(* IEC 61131-3 sources: moqui-plc/agent-skills/output/sessions/demo-plant-session/generated-plc/demo-hvac/src/main/org/moqui/device, 4 files *)

(* ---- DeviceFacade.dut ---- *)
(*
 * DeviceFacade implementation for managing devices and logical parameters.
 *
 * Naming rules:
 *   deviceName + parameterName or parameterName -> logical signal
 *   deviceName + parameterName or parameterName + Min/Max -> limits
 *
 * All digital signals (boolean) are active-high (positive logic).
 * All durations are expressed in seconds TUnit.
 *)
TYPE DeviceFacade : STRUCT
    (* ========== Analog process/environment parameters ========== *)
    (* TODO: declare REAL process/environment parameters *)

    (* ========== Digital process/environment parameters ========== *)
    (* TODO: declare BOOL process/environment parameters *)

    (* Boolean predicates - computed each scan by MainRuleEngine *)
    (* TODO: declare computed predicates used by MainRuleEngine *)

    (* Operating-mode flags and process timing (mapped from recipe). *)
    estimatedRuntime : TUnit;
    minRuntime : TUnit;
    estimatedBreakDuration : TUnit;
    minBreakDuration : TUnit;
    processEstimatedDuration : TUnit;
    processMinDuration : TUnit;
    processActualDuration : TUnit;
    processRemainingDuration : TUnit;
    actualRuntime : TUnit;
    actualBreakDuration : TUnit;
    timeBreakEnabled : BOOL;
    isCompleted : BOOL;

    (* Main FSM state and transition request/acknowledge commands *)
    status : MainStatus := MainStatus.Disabled;
    lastStatus : MainStatus := MainStatus.Disabled;
    disabledRequest : BOOL;
    standstillRequest : BOOL;
    homingRequest : BOOL;
    runRequest : BOOL;
    synchronizedRunRequest : BOOL;
    stoppingRequest : BOOL;
    errorStopRequest : BOOL;
    faultRequest : BOOL;
    faultAck : BOOL;

    (* ========== Atomic devices ========== *)
    (* TODO: declare Actuator/ActuatorGroup/Axis/AxisGroup/ProcessPid instances *)

    (* Signal management - centralised fault / alarm / warning engine *)
    signalMgmt : SignalMgmt;
END_STRUCT END_TYPE

(* Questions for the skill/user:
 * 1. Which analog input signals and setpoints must be declared as REAL?
 * 2. Which digital signals must be declared as BOOL?
 * 3. Which computed predicates are required by MainRuleEngine?
 * 4. Which timing/process flags are needed (estimatedRuntime, minRuntime, etc.)?
 * 5. Which request flags correspond to the states in the selected StatusFlow?
 * 6. Which atomic devices exist: Actuator, ActuatorGroup, Axis, AxisGroup, ProcessPid?
 *)

(* ---- IOFacade.dut ---- *)
(*
 * IOFacade implementation for managing physical devices and input/output signals/terminals.
 * Input/Output physical terminals naming rules.
 * From each value of the Parameter entity 3 signals will be generated, according to the following naming convention:
 *     deviceName + parameterName or parameterName + physicalAddress (e.g.: Channel + PhysicalAddress for Modbus)
 *     deviceName + parameterName or parameterName + Min/Max + physicalAddress (e.g.: Channel + PhysicalAddress for Modbus)
 *
 * The physicalAdddress suffix will have the following syntax:
 *    %<memory area prefix> ( <size prefix> )? <memory position>
 * where
 *    <memory area prefix> : I | Q | M
 *    <size prefix> : X | B | W | D
 *    <memory position> : <number> ( .<number> )* (* Depends on the target system *)
 *
 * An alternative is to use semantic signal naming rules.
 *)
TYPE IOFacade : STRUCT
    (* ========== Phyisical Input Terminals/Signals ========== *)
    (* TODO: declare physical input signals from DeviceRequestItem or naming convention *)

    (* ========== Phyisical Output Terminals/Signals ========== *)
    (* TODO: declare physical output signals from DeviceRequestItem or naming convention *)
END_STRUCT END_TYPE

(* Generation notes:
 * - This file is auto-generable from DeviceRequestItem metadata or from naming conventions.
 * - The logical-to-physical mapping remains outside this template and stays manual in V1.
 *
 * Questions for the skill/user:
 * 1. Should names come from DeviceRequestItem.requestItemName or from naming conventions?
 * 2. Which physical signals are inputs and which are outputs?
 * 3. What IEC type should be used for each signal?
 * 4. Are there address-based names, semantic names, or both?
 *)

(* ---- DeviceDiagnostics.pou ---- *)
{attribute 'no_assign'}
(* Device diagnostics *)
FUNCTION_BLOCK DeviceDiagnostics
VAR_EXTERNAL
    dev : DeviceFacade;
END_VAR
VAR_INPUT
    operationType : OperatingMode := OperatingMode.Run;
END_VAR
VAR_OUTPUT
    error : BOOL;
END_VAR

error := TRUE;

(* Signal management engine *)
(*
 * Prepare a fresh scan (clears the accumulated output action).
 * Then process each device signal in priority order.
 * ImmediateStop -> faultRequest := TRUE -> Main enters Fault state.
 *)
dev.signalMgmt(operationType := SignalMgmtOperatingMode.Prepare);
dev.signalMgmt.operationType := SignalMgmtOperatingMode.Process;

(* Device faults *)
(* TODO: add blocking device diagnostics rules *)

(* Environmental / safety diagnostics *)
(* TODO: add environmental and safety stop rules *)

error := FALSE;

(* Questions for the skill/user:
 * 1. Which device faults are blocking and must trigger ImmediateStop?
 * 2. For each blocking device, which signal should be monitored:
 *    fault, invalidConfig, cmdError, externalFault, etc.?
 * 3. Which environmental/safety predicates should become alarms?
 * 4. Which predicates are warnings only and should not stop the machine?
 *)

(* ---- DeviceManager.pou ---- *)
{attribute 'no_assign'}
(* Hardware Abstraction Layer (HAL) orchestrator.
 *
 * Drives all physical device FBs once per scan.
 * Main component sets the enable/disable request flags; DeviceManager wires them
 * to the individual Actuator / ProcessPid FBs.
 *
 * Call order within the PLC task:
 *   InputSignalUpdate (updates feedback signals from field)
 *   Main (FSM + DeviceRuleEngine -> sets request flags)
 *   DeviceManager (this block - drives device FBs)
 *   OutputSignalUpdate (maps device outputs to physical terminals)
 *
 * Handshake note (Actuator FBs):
 *   enableRequest / disableRequest are VAR_IN_OUT.  The Actuator FB clears
 *   the flag as its acknowledgment.  Main.pou re-asserts the flag each scan
 *   from dev.xxxEnableRequest, so the handshake is level-triggered.
 *
 * ProcessPid note (ahuFan):
 *   ProcessPid uses a plain BOOL 'enable' input - no VAR_IN_OUT handshake.
 *   Setting enable := FALSE ramps the output to 0 and disables the controller.
 *)
FUNCTION_BLOCK DeviceManager
VAR_EXTERNAL
    clks : Clocks;
    dev : DeviceFacade;
END_VAR
VAR_INPUT
    operationType : OperatingMode := OperatingMode.Run;
END_VAR

(* Atomic device orchestration *)
(* TODO: invoke each atomic device instance in deterministic order *)

(* Questions for the skill/user:
 * 1. Which atomic devices must be called every scan?
 * 2. For each Actuator, which enableRequest/disableRequest flags drive it?
 * 3. For each ProcessPid, which enable/setpoint/feedback signals drive it?
 * 4. For each Axis or AxisGroup, which command/enable structures are used?
 *)
